TYPE E_OpClCtrl :
(
	Open,
	Close
)USINT;
END_TYPE

(* stored: Version 1.1.0.1, ProductVersion 3.1.0.25
   DUT E_OpClCtrl: Id {1fb760e4-9ee5-4fde-953d-c69117ebd443} *)
